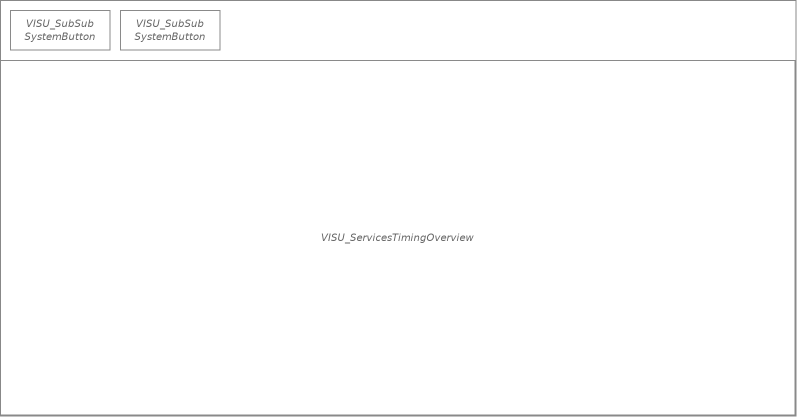
VISUALIZATION VISU_ServicesTiming  // 797x417
VAR_IN_OUT
	ref : ServicesTiming;
    widget : ServicesTimingWidget;
END_VAR
    Frame (10,10 100x40)
        shows VISU_SubSubSystemButton(widget := widget.button_overview)
    Frame (120,10 100x40)
        shows VISU_SubSubSystemButton(widget := widget.button_io)
    Frame (0,60 795x355), frame switch variable: widget.activeTab
        shows VISU_ServicesTimingOverview(ref := ref, widget := widget)
        shows VISU_ServicesTimingIO(ref := ref.parts.io, widget := widget.io)
END_VISUALIZATION

(* stored: Version 1.1.0.1, ProductVersion 3.1.4019.2
   Visu VISU_ServicesTiming: Id {353b08a7-bad0-42b8-bf15-fe60483bce8f} *)
